TYPE st_Networking :
STRUCT
	b_MaintenanceWifiActive	:	BOOL
	ui_
END_STRUCT
END_TYPE

(* stored: Version 1.1.0.1, ProductVersion 3.1.4024.12
   DUT st_Networking: Id {e2d2018c-a73c-459c-89d1-e77e2b5d7b33} *)
